(* PLC project Tc2_Utilities.WritePersistentData Demo, tc3-libraries-kb TwinCAT 3.1 *)
(* stored: creationDateTime 2026-05-11T00:00:00, modificationDateTime 2026-05-11T00:00:00 *)

PROGRAM P_Demo_WritePersistentData
  VAR
    fbWritePersistentData : WritePersistentData;  (* WritePersistentData 实例 *)
    bWrite : BOOL := FALSE;
    bBusy_ : BOOL;
    bErrFlag : BOOL;
    nErrCode : UDINT;
  END_VAR

// =============================================================================
// 场景：兼容旧项目。
// 价值：向后兼容。
// 验证：同 FB_WritePersistentData。
// 验证步骤：
//   1. 右键 PLC 项目 → Import PLCopenXML → 选本文件
//   2. 引用 Tc2_Utilities（References → Add library）
//   3. 编译 → 登录 → 运行；按上方『验证』行的指示在线写值观察
// =============================================================================

fbWritePersistentData(
    NETID := '', PORT := 851, START := bWrite, TMOUT := DEFAULT_ADS_TIMEOUT,
    BUSY => bBusy_, ERR => bErrFlag, ERRID => nErrCode
);
END_PROGRAM
